FUNCTION_BLOCK ConveyorRenderTwoConveyor (* Basic Function Block Type *)
  (* Standard: 61499-2 *)
  (* Version 0.2, 2003-12-04, JHC, Rockwell Automation, Renamed for better indexing. *)
  (* Version 0.1, 2002-11-05, JHC, Rockwell Automation, Corrected missing ST element in Algorithm REQ. *)
  (* Version 0.0, 2000-05-30, JHC, Rockwell Automation *)
  (* Compiler header: package fb.rt.cs725; *)
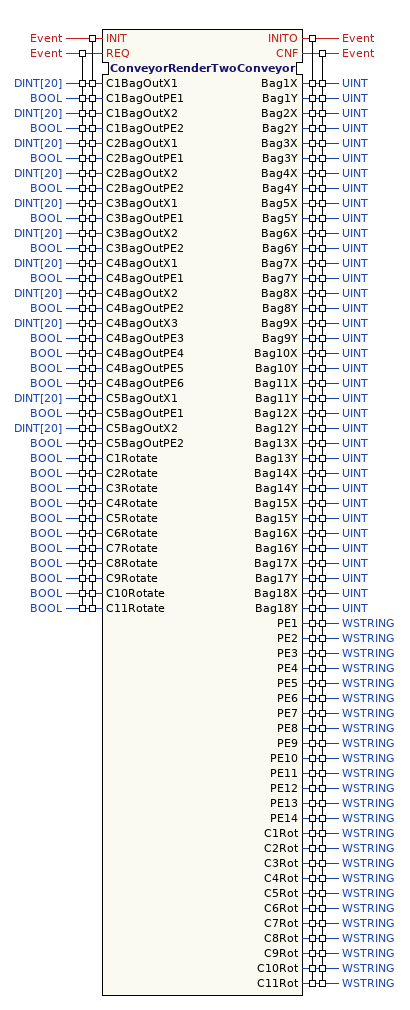
  EVENT_INPUT
    INIT WITH C1BagOutX1, C1BagOutPE1, C1BagOutX2, C1BagOutPE2, C2BagOutX1, C2BagOutPE1, C2BagOutX2, C2BagOutPE2, C3BagOutX1, C3BagOutPE1, C3BagOutX2, C3BagOutPE2, C4BagOutX1, C4BagOutPE1, C4BagOutX2, C4BagOutPE2, C4BagOutX3, C4BagOutPE3, C4BagOutPE5, C4BagOutPE4, C1Rotate, C2Rotate, C3Rotate, C4Rotate, C5Rotate, C6Rotate, C7Rotate, C8Rotate, C9Rotate, C10Rotate, C11Rotate, C4BagOutPE6, C5BagOutX1, C5BagOutPE1, C5BagOutX2, C5BagOutPE2; (* Initialization Request *)
    REQ WITH C1BagOutX1, C1BagOutPE1, C1BagOutX2, C1BagOutPE2, C2BagOutX1, C2BagOutPE1, C2BagOutX2, C2BagOutPE2, C3BagOutX1, C3BagOutPE1, C3BagOutX2, C3BagOutPE2, C4BagOutX1, C4BagOutPE1, C4BagOutX2, C4BagOutPE2, C4BagOutX3, C4BagOutPE3, C4BagOutPE4, C4BagOutPE5, C1Rotate, C2Rotate, C3Rotate, C4Rotate, C5Rotate, C6Rotate, C7Rotate, C8Rotate, C9Rotate, C10Rotate, C11Rotate, C4BagOutPE6, C5BagOutX1, C5BagOutPE1, C5BagOutX2, C5BagOutPE2; (* Normal Execution Request *)
  END_EVENT
  EVENT_OUTPUT
    INITO WITH Bag1X, Bag1Y, Bag2X, Bag2Y, Bag3X, Bag3Y, Bag4X, Bag4Y, Bag5X, Bag5Y, Bag6X, Bag6Y, Bag7X, Bag7Y, Bag8X, Bag8Y, Bag9X, Bag9Y, Bag10X, Bag10Y, Bag11X, Bag11Y, Bag12X, Bag12Y, Bag13X, Bag13Y, Bag14X, Bag14Y, Bag15X, Bag15Y, Bag16X, Bag16Y, Bag17X, Bag17Y, Bag18X, Bag18Y, PE1, PE2, PE3, PE4, PE5, PE6, PE7, PE8, PE9, PE10, PE11, PE12, PE13, PE14, C1Rot, C2Rot, C3Rot, C4Rot, C5Rot, C6Rot, C7Rot, C8Rot, C9Rot, C10Rot, C11Rot; (* Initialization Confirm *)
    CNF WITH Bag1X, Bag1Y, Bag2X, Bag2Y, Bag3X, Bag3Y, Bag4X, Bag4Y, Bag5X, Bag5Y, Bag6X, Bag6Y, Bag7X, Bag7Y, Bag8X, Bag8Y, Bag9X, Bag9Y, Bag10X, Bag10Y, Bag11X, Bag11Y, Bag12X, Bag12Y, Bag13X, Bag13Y, Bag14X, Bag14Y, Bag15X, Bag15Y, Bag16X, Bag16Y, Bag17X, Bag17Y, Bag18X, Bag18Y, PE1, PE2, PE3, PE4, PE5, PE6, PE7, PE8, PE9, PE10, PE11, PE12, PE13, PE14, C1Rot, C2Rot, C3Rot, C4Rot, C5Rot, C6Rot, C7Rot, C8Rot, C9Rot, C10Rot, C11Rot; (* Execution Confirmation *)
  END_EVENT
  VAR_INPUT
    C1BagOutX1 : ARRAY [0..19] OF DINT;
    C1BagOutPE1 : BOOL;
    C1BagOutX2 : ARRAY [0..19] OF DINT;
    C1BagOutPE2 : BOOL;
    C2BagOutX1 : ARRAY [0..19] OF DINT;
    C2BagOutPE1 : BOOL;
    C2BagOutX2 : ARRAY [0..19] OF DINT;
    C2BagOutPE2 : BOOL;
    C3BagOutX1 : ARRAY [0..19] OF DINT;
    C3BagOutPE1 : BOOL;
    C3BagOutX2 : ARRAY [0..19] OF DINT;
    C3BagOutPE2 : BOOL;
    C4BagOutX1 : ARRAY [0..19] OF DINT;
    C4BagOutPE1 : BOOL;
    C4BagOutX2 : ARRAY [0..19] OF DINT;
    C4BagOutPE2 : BOOL;
    C4BagOutX3 : ARRAY [0..19] OF DINT;
    C4BagOutPE3 : BOOL;
    C4BagOutPE4 : BOOL;
    C4BagOutPE5 : BOOL;
    C4BagOutPE6 : BOOL;
    C5BagOutX1 : ARRAY [0..19] OF DINT;
    C5BagOutPE1 : BOOL;
    C5BagOutX2 : ARRAY [0..19] OF DINT;
    C5BagOutPE2 : BOOL;
    C1Rotate : BOOL;
    C2Rotate : BOOL;
    C3Rotate : BOOL;
    C4Rotate : BOOL;
    C5Rotate : BOOL;
    C6Rotate : BOOL;
    C7Rotate : BOOL;
    C8Rotate : BOOL;
    C9Rotate : BOOL;
    C10Rotate : BOOL;
    C11Rotate : BOOL;
  END_VAR
  VAR_OUTPUT
    Bag1X : UINT;
    Bag1Y : UINT;
    Bag2X : UINT;
    Bag2Y : UINT;
    Bag3X : UINT;
    Bag3Y : UINT;
    Bag4X : UINT;
    Bag4Y : UINT;
    Bag5X : UINT;
    Bag5Y : UINT;
    Bag6X : UINT;
    Bag6Y : UINT;
    Bag7X : UINT;
    Bag7Y : UINT;
    Bag8X : UINT;
    Bag8Y : UINT;
    Bag9X : UINT;
    Bag9Y : UINT;
    Bag10X : UINT;
    Bag10Y : UINT;
    Bag11X : UINT;
    Bag11Y : UINT;
    Bag12X : UINT;
    Bag12Y : UINT;
    Bag13X : UINT;
    Bag13Y : UINT;
    Bag14X : UINT;
    Bag14Y : UINT;
    Bag15X : UINT;
    Bag15Y : UINT;
    Bag16X : UINT;
    Bag16Y : UINT;
    Bag17X : UINT;
    Bag17Y : UINT;
    Bag18X : UINT;
    Bag18Y : UINT;
    PE1 : WSTRING;
    PE2 : WSTRING;
    PE3 : WSTRING;
    PE4 : WSTRING;
    PE5 : WSTRING;
    PE6 : WSTRING;
    PE7 : WSTRING;
    PE8 : WSTRING;
    PE9 : WSTRING;
    PE10 : WSTRING;
    PE11 : WSTRING;
    PE12 : WSTRING;
    PE13 : WSTRING;
    PE14 : WSTRING;
    C1Rot : WSTRING;
    C2Rot : WSTRING;
    C3Rot : WSTRING;
    C4Rot : WSTRING;
    C5Rot : WSTRING;
    C6Rot : WSTRING;
    C7Rot : WSTRING;
    C8Rot : WSTRING;
    C9Rot : WSTRING;
    C10Rot : WSTRING;
    C11Rot : WSTRING;
  END_VAR
  VAR
    numOfBags : INT := 0;
    index : INT := 0;
    bagDetail : ARRAY [0..17] OF BagDetail;
    tcOffset1 : INT;
    tcOffset2 : INT;
    tcOffset3 : INT;
    fcOffset1 : INT;
    fcOffset2 : INT;
    fc1Offset1 : INT;
    fc1Offset2 : INT;
    fc2Offset1 : INT;
    fc2Offset2 : INT;
  END_VAR
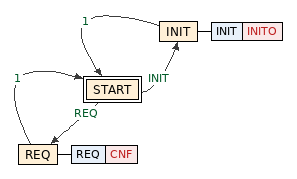
  EC_STATES
    START; (* Initial State *)
    INIT : INIT -> INITO; (* Initialization *)
    REQ : REQ -> CNF; (* Normal execution *)
  END_STATES
  EC_TRANSITIONS
    START TO INIT := INIT;
    INIT TO START := 1;
    START TO REQ := REQ;
    REQ TO START := 1;
  END_TRANSITIONS
  ALGORITHM INIT IN Java: (* Initialization algorithm *)
Bag1X.value=6000;
Bag1Y.value=6000;
Bag2X.value=6000;
Bag2Y.value=6000;
Bag3X.value=6000;
Bag3Y.value=6000;
Bag4X.value=6000;
Bag4Y.value=6000;
Bag5X.value=6000;
Bag5Y.value=6000;
Bag6X.value=6000;
Bag6Y.value=6000;
Bag7X.value=6000;
Bag7Y.value=6000;
Bag8X.value=6000;
Bag8Y.value=6000;
Bag9X.value=6000;
Bag9Y.value=6000;
Bag10X.value=6000;
Bag10Y.value=6000;
Bag11X.value=6000;
Bag11Y.value=6000;
Bag12X.value=6000;
Bag12Y.value=6000;
Bag13X.value=6000;
Bag13Y.value=6000;
Bag14X.value=6000;
Bag14Y.value=6000;
Bag15X.value=6000;
Bag15Y.value=6000;
Bag16X.value=6000;
Bag16Y.value=6000;
Bag17X.value=6000;
Bag17Y.value=6000;
Bag18X.value=6000;
Bag18Y.value=6000;


for(int i = 0; i < 18; i++)
{
    ((BagDetail)bagDetail.value[i]).bagYValue.value=6000;
    ((BagDetail)bagDetail.value[i]).conId.value=6000;
    ((BagDetail)bagDetail.value[i]).bagXValue.value=6000;
}

fcOffset1.value=49;
fcOffset2.value=201;
fc1Offset1.value=659;
fc1Offset2.value=507;
fc2Offset1.value=659;
fc2Offset2.value=507;
tcOffset1.value=99;
tcOffset2.value=301;
tcOffset3.value=503;
if (C1BagOutPE1.value)
PE1.value = "/fb/rt/cs725/SSG.png";
else
PE1.value = "/fb/rt/cs725/SSR.png";
if (C1BagOutPE2.value)
PE2.value = "/fb/rt/cs725/SSG.png";
else
PE2.value = "/fb/rt/cs725/SSR.png";

if (C2BagOutPE1.value)
PE3.value = "/fb/rt/cs725/SSG.png";
else
PE3.value = "/fb/rt/cs725/SSR.png";
if (C2BagOutPE2.value)
PE4.value = "/fb/rt/cs725/SSG.png";
else
PE4.value = "/fb/rt/cs725/SSR.png";

if (C3BagOutPE1.value)
PE5.value = "/fb/rt/cs725/SSG.png";
else
PE5.value = "/fb/rt/cs725/SSR.png";
if (C3BagOutPE2.value)
PE6.value = "/fb/rt/cs725/SSG.png";
else
PE6.value = "/fb/rt/cs725/SSR.png";

if (C4BagOutPE1.value)
PE7.value = "/fb/rt/cs725/SSG.png";
else
PE7.value = "/fb/rt/cs725/SSR.png";
if (C4BagOutPE2.value)
PE8.value = "/fb/rt/cs725/SSG.png";
else
PE8.value = "/fb/rt/cs725/SSR.png";
if (C4BagOutPE3.value)
PE9.value = "/fb/rt/cs725/SSG.png";
else
PE9.value = "/fb/rt/cs725/SSR.png";
if (C4BagOutPE4.value)
PE10.value = "/fb/rt/cs725/SSG.png";
else
PE10.value = "/fb/rt/cs725/SSR.png";
if (C4BagOutPE5.value)
PE11.value = "/fb/rt/cs725/SSG.png";
else
PE11.value = "/fb/rt/cs725/SSR.png";
if (C4BagOutPE6.value)
PE12.value = "/fb/rt/cs725/SSG.png";
else
PE12.value = "/fb/rt/cs725/SSR.png";

if (C5BagOutPE1.value)
PE13.value = "/fb/rt/cs725/SSG.png";
else
PE13.value = "/fb/rt/cs725/SSR.png";
if (C5BagOutPE2.value)
PE14.value = "/fb/rt/cs725/SSG.png";
else
PE14.value = "/fb/rt/cs725/SSR.png";

if (C1Rotate.value)
C1Rot.value = "/fb/rt/cs725/FC.gif";
else
C1Rot.value = "/fb/rt/cs725/FC.png";

if (C2Rotate.value)
C2Rot.value = "/fb/rt/cs725/FC.gif";
else
C2Rot.value = "/fb/rt/cs725/FC.png";

if (C3Rotate.value)
C3Rot.value = "/fb/rt/cs725/FC.gif";
else
C3Rot.value = "/fb/rt/cs725/FC.png";

if (C4Rotate.value)
C4Rot.value = "/fb/rt/cs725/FC.gif";
else
C4Rot.value = "/fb/rt/cs725/FC.png";

if (C5Rotate.value)
C5Rot.value = "/fb/rt/cs725/FCU.gif";
else
C5Rot.value = "/fb/rt/cs725/FCU.png";

if (C6Rotate.value)
C6Rot.value = "/fb/rt/cs725/FCU.gif";
else
C6Rot.value = "/fb/rt/cs725/FCU.png";

if (C7Rotate.value)
C7Rot.value = "/fb/rt/cs725/TC.gif";
else
C7Rot.value = "/fb/rt/cs725/TC.png";

if (C8Rotate.value)
C8Rot.value = "/fb/rt/cs725/TC.gif";
else
C8Rot.value = "/fb/rt/cs725/TC.png";

if (C9Rotate.value)
C9Rot.value = "/fb/rt/cs725/TC.gif";
else
C9Rot.value = "/fb/rt/cs725/TC.png";

if (C10Rotate.value)
C10Rot.value = "/fb/rt/cs725/FCU.gif";
else
C10Rot.value = "/fb/rt/cs725/FCU.png";

if (C11Rotate.value)
C11Rot.value = "/fb/rt/cs725/FCU.gif";
else
C11Rot.value = "/fb/rt/cs725/FCU.png";
  END_ALGORITHM
  ALGORITHM REQ IN Java: (* Normally executed algorithm *)
index.value=0;

for(int i = 0; i < 5 ; i++)
{
  if(index.value < 16)
  {

    if(((DINT)C1BagOutX1.value[i]).value != 0)
    {
        ((BagDetail)bagDetail.value[index.value]).conId.value=1;
((BagDetail)bagDetail.value[index.value]).bagYValue.value=fcOffset1.value+((DINT)C1BagOutX1.value[i]).value;
index.value++;
    }
    if(((DINT)C1BagOutX2.value[i]).value != 0)
    {

        ((BagDetail)bagDetail.value[index.value]).conId.value=1;
((BagDetail)bagDetail.value[index.value]).bagYValue.value=fcOffset2.value+((DINT)C1BagOutX2.value[i]).value;
index.value++;
    }
    if(((DINT)C2BagOutX1.value[i]).value != 0)
    {
        ((BagDetail)bagDetail.value[index.value]).conId.value=2;
((BagDetail)bagDetail.value[index.value]).bagYValue.value=fcOffset1.value+((DINT)C2BagOutX1.value[i]).value;
index.value++;
    }
    if(((DINT)C2BagOutX2.value[i]).value != 0)
    {
        ((BagDetail)bagDetail.value[index.value]).conId.value=2;
((BagDetail)bagDetail.value[index.value]).bagYValue.value=fcOffset2.value+((DINT)C2BagOutX2.value[i]).value;
index.value++;
    }
    if(((DINT)C3BagOutX1.value[i]).value != 0)
    {
        ((BagDetail)bagDetail.value[index.value]).conId.value=3;
((BagDetail)bagDetail.value[index.value]).bagYValue.value=fc1Offset1.value-((DINT)C3BagOutX1.value[i]).value;
index.value++;
    }
    if(((DINT)C3BagOutX2.value[i]).value != 0)
    {
        ((BagDetail)bagDetail.value[index.value]).conId.value=3;
((BagDetail)bagDetail.value[index.value]).bagYValue.value=fc1Offset2.value-((DINT)C3BagOutX2.value[i]).value;
index.value++;
    }
    if(((DINT)C5BagOutX1.value[i]).value != 0)
    {
        ((BagDetail)bagDetail.value[index.value]).conId.value=4;
((BagDetail)bagDetail.value[index.value]).bagYValue.value=fc2Offset1.value-((DINT)C5BagOutX1.value[i]).value;
index.value++;
    }
    if(((DINT)C5BagOutX2.value[i]).value != 0)
    {
        ((BagDetail)bagDetail.value[index.value]).conId.value=4;
((BagDetail)bagDetail.value[index.value]).bagYValue.value=fc2Offset2.value-((DINT)C5BagOutX2.value[i]).value;
index.value++;
    }
 }
}
for(int i = 0; i < 16 ; i++)
{
  if(index.value < 16)
  {
    if(((DINT)C4BagOutX1.value[i]).value != 0)
    {
        ((BagDetail)bagDetail.value[index.value]).conId.value=0;
((BagDetail)bagDetail.value[index.value]).bagXValue.value=tcOffset1.value+((DINT)C4BagOutX1.value[i]).value;
index.value++;
    }
    if(((DINT)C4BagOutX2.value[i]).value != 0)
    {
        ((BagDetail)bagDetail.value[index.value]).conId.value=0;
((BagDetail)bagDetail.value[index.value]).bagXValue.value=tcOffset2.value+((DINT)C4BagOutX2.value[i]).value;
index.value++;
    }
    if(((DINT)C4BagOutX3.value[i]).value != 0)
    {
        ((BagDetail)bagDetail.value[index.value]).conId.value=0;
((BagDetail)bagDetail.value[index.value]).bagXValue.value=tcOffset3.value+((DINT)C4BagOutX3.value[i]).value;
index.value++;
    }
  }
}
for(int i = 0; i < 16; i++)
{
    switch(((BagDetail)bagDetail.value[i]).conId.value)
{
case 0: ((BagDetail)bagDetail.value[i]).bagYValue.value = 359;
        break;
case 1:((BagDetail)bagDetail.value[i]).bagXValue.value = 105;
        break;
case 2:((BagDetail)bagDetail.value[i]).bagXValue.value = 307;
        break;
case 3:((BagDetail)bagDetail.value[i]).bagXValue.value = 205;
        break;
case 4:((BagDetail)bagDetail.value[i]).bagXValue.value = 509;
        break;
case 6000: ((BagDetail)bagDetail.value[i]).bagXValue.value = 6000;
           ((BagDetail)bagDetail.value[i]).bagYValue.value = 6000;
        break;
}
}
Bag1X.value=6000;
Bag1Y.value=6000;
Bag2X.value=6000;
Bag2Y.value=6000;
Bag3X.value=6000;
Bag3Y.value=6000;
Bag4X.value=6000;
Bag4Y.value=6000;
Bag5X.value=6000;
Bag5Y.value=6000;
Bag6X.value=6000;
Bag6Y.value=6000;
Bag7X.value=6000;
Bag7Y.value=6000;
Bag8X.value=6000;
Bag8Y.value=6000;
Bag9X.value=6000;
Bag9Y.value=6000;
Bag10X.value=6000;
Bag10Y.value=6000;
Bag11X.value=6000;
Bag11Y.value=6000;
Bag12X.value=6000;
Bag12Y.value=6000;
Bag13X.value=6000;
Bag13Y.value=6000;
Bag14X.value=6000;
Bag14Y.value=6000;
Bag15X.value=6000;
Bag15Y.value=6000;
Bag16X.value=6000;
Bag16Y.value=6000;
Bag17X.value=6000;
Bag17Y.value=6000;
Bag18X.value=6000;
Bag18Y.value=6000;
for(int i = 0; i < 16; i++)
{
    switch(i)
        {
           case 0: Bag1X.value = ((BagDetail)bagDetail.value[i]).bagXValue.value;
           Bag1Y.value = ((BagDetail)bagDetail.value[i]).bagYValue.value;
   break;
   case 1: Bag2X.value = ((BagDetail)bagDetail.value[i]).bagXValue.value;
           Bag2Y.value = ((BagDetail)bagDetail.value[i]).bagYValue.value;
   break;
   case 2: Bag3X.value = ((BagDetail)bagDetail.value[i]).bagXValue.value;
           Bag3Y.value = ((BagDetail)bagDetail.value[i]).bagYValue.value;
   break;
   case 3: Bag4X.value = ((BagDetail)bagDetail.value[i]).bagXValue.value;
           Bag4Y.value = ((BagDetail)bagDetail.value[i]).bagYValue.value;
   break;
   case 4: Bag5X.value = ((BagDetail)bagDetail.value[i]).bagXValue.value;
           Bag5Y.value = ((BagDetail)bagDetail.value[i]).bagYValue.value;
   break;
   case 5: Bag6X.value = ((BagDetail)bagDetail.value[i]).bagXValue.value;
           Bag6Y.value = ((BagDetail)bagDetail.value[i]).bagYValue.value;
   break;
   case 6: Bag7X.value = ((BagDetail)bagDetail.value[i]).bagXValue.value;
           Bag7Y.value = ((BagDetail)bagDetail.value[i]).bagYValue.value;
   break;
   case 7: Bag8X.value = ((BagDetail)bagDetail.value[i]).bagXValue.value;
           Bag8Y.value = ((BagDetail)bagDetail.value[i]).bagYValue.value;
   break;
   case 8: Bag9X.value = ((BagDetail)bagDetail.value[i]).bagXValue.value;
           Bag9Y.value = ((BagDetail)bagDetail.value[i]).bagYValue.value;
   break;
   case 9: Bag10X.value = ((BagDetail)bagDetail.value[i]).bagXValue.value;
           Bag10Y.value = ((BagDetail)bagDetail.value[i]).bagYValue.value;
   break;
case 10: Bag11X.value = ((BagDetail)bagDetail.value[i]).bagXValue.value;
           Bag11Y.value = ((BagDetail)bagDetail.value[i]).bagYValue.value;
   break;
   case 11: Bag12X.value = ((BagDetail)bagDetail.value[i]).bagXValue.value;
           Bag12Y.value = ((BagDetail)bagDetail.value[i]).bagYValue.value;
   break;
   case 12: Bag13X.value = ((BagDetail)bagDetail.value[i]).bagXValue.value;
           Bag13Y.value = ((BagDetail)bagDetail.value[i]).bagYValue.value;
   break;
   case 13: Bag14X.value = ((BagDetail)bagDetail.value[i]).bagXValue.value;
           Bag14Y.value = ((BagDetail)bagDetail.value[i]).bagYValue.value;
   break;
   case 14: Bag15X.value = ((BagDetail)bagDetail.value[i]).bagXValue.value;
           Bag15Y.value = ((BagDetail)bagDetail.value[i]).bagYValue.value;
   break;
   case 15: Bag16X.value = ((BagDetail)bagDetail.value[i]).bagXValue.value;
           Bag16Y.value = ((BagDetail)bagDetail.value[i]).bagYValue.value;
   break;
   case 16: Bag17X.value = ((BagDetail)bagDetail.value[i]).bagXValue.value;
           Bag17Y.value = ((BagDetail)bagDetail.value[i]).bagYValue.value;
   break;
   case 17: Bag18X.value = ((BagDetail)bagDetail.value[i]).bagXValue.value;
           Bag18Y.value = ((BagDetail)bagDetail.value[i]).bagYValue.value;
   break;
    }
}


for(int i = 0; i < 10; i++)
{
    ((BagDetail)bagDetail.value[i]).bagYValue.value=6000;
    ((BagDetail)bagDetail.value[i]).conId.value=6000;
    ((BagDetail)bagDetail.value[i]).bagXValue.value=6000;
}

if (C1BagOutPE1.value)
PE1.value = "/fb/rt/cs725/SSG.png";
else
PE1.value = "/fb/rt/cs725/SSR.png";
if (C1BagOutPE2.value)
PE2.value = "/fb/rt/cs725/SSG.png";
else
PE2.value = "/fb/rt/cs725/SSR.png";

if (C2BagOutPE1.value)
PE3.value = "/fb/rt/cs725/SSG.png";
else
PE3.value = "/fb/rt/cs725/SSR.png";
if (C2BagOutPE2.value)
PE4.value = "/fb/rt/cs725/SSG.png";
else
PE4.value = "/fb/rt/cs725/SSR.png";

if (C3BagOutPE1.value)
PE5.value = "/fb/rt/cs725/SSG.png";
else
PE5.value = "/fb/rt/cs725/SSR.png";
if (C3BagOutPE2.value)
PE6.value = "/fb/rt/cs725/SSG.png";
else
PE6.value = "/fb/rt/cs725/SSR.png";

if (C4BagOutPE1.value)
PE7.value = "/fb/rt/cs725/SSG.png";
else
PE7.value = "/fb/rt/cs725/SSR.png";
if (C4BagOutPE2.value)
PE8.value = "/fb/rt/cs725/SSG.png";
else
PE8.value = "/fb/rt/cs725/SSR.png";
if (C4BagOutPE3.value)
PE9.value = "/fb/rt/cs725/SSG.png";
else
PE9.value = "/fb/rt/cs725/SSR.png";
if (C4BagOutPE4.value)
PE10.value = "/fb/rt/cs725/SSG.png";
else
PE10.value = "/fb/rt/cs725/SSR.png";
if (C4BagOutPE5.value)
PE11.value = "/fb/rt/cs725/SSG.png";
else
PE11.value = "/fb/rt/cs725/SSR.png";
if (C4BagOutPE6.value)
PE12.value = "/fb/rt/cs725/SSG.png";
else
PE12.value = "/fb/rt/cs725/SSR.png";

if (C5BagOutPE1.value)
PE13.value = "/fb/rt/cs725/SSG.png";
else
PE13.value = "/fb/rt/cs725/SSR.png";
if (C5BagOutPE2.value)
PE14.value = "/fb/rt/cs725/SSG.png";
else
PE14.value = "/fb/rt/cs725/SSR.png";

if (C1Rotate.value)
C1Rot.value = "/fb/rt/cs725/FC.gif";
else
C1Rot.value = "/fb/rt/cs725/FC.png";

if (C2Rotate.value)
C2Rot.value = "/fb/rt/cs725/FC.gif";
else
C2Rot.value = "/fb/rt/cs725/FC.png";

if (C3Rotate.value)
C3Rot.value = "/fb/rt/cs725/FC.gif";
else
C3Rot.value = "/fb/rt/cs725/FC.png";

if (C4Rotate.value)
C4Rot.value = "/fb/rt/cs725/FC.gif";
else
C4Rot.value = "/fb/rt/cs725/FC.png";

if (C5Rotate.value)
C5Rot.value = "/fb/rt/cs725/FCU.gif";
else
C5Rot.value = "/fb/rt/cs725/FCU.png";

if (C6Rotate.value)
C6Rot.value = "/fb/rt/cs725/FCU.gif";
else
C6Rot.value = "/fb/rt/cs725/FCU.png";

if (C7Rotate.value)
C7Rot.value = "/fb/rt/cs725/TC.gif";
else
C7Rot.value = "/fb/rt/cs725/TC.png";

if (C8Rotate.value)
C8Rot.value = "/fb/rt/cs725/TC.gif";
else
C8Rot.value = "/fb/rt/cs725/TC.png";

if (C9Rotate.value)
C9Rot.value = "/fb/rt/cs725/TC.gif";
else
C9Rot.value = "/fb/rt/cs725/TC.png";

if (C10Rotate.value)
C10Rot.value = "/fb/rt/cs725/FCU.gif";
else
C10Rot.value = "/fb/rt/cs725/FCU.png";

if (C11Rotate.value)
C11Rot.value = "/fb/rt/cs725/FCU.gif";
else
C11Rot.value = "/fb/rt/cs725/FCU.png";
  END_ALGORITHM
  ALGORITHM BAGIN IN Java:
//if(numOfBags.value < 10)
{
  // numOfBags.value++;
}
  END_ALGORITHM
END_FUNCTION_BLOCK
